// TIA Portal V20 export
TYPE "typeFDoorSignal"
// Safety status of door
// stored: Access Published, IsFailsafeCompliant true, Namespace Safety
   STRUCT
      reqDoorUnlock1 : Bool;   // Cmd Maint Door1 Open Request
      reqDoorUnlock2 : Bool;   // Cmd Maint Door2 Open Request
      reqDoorUnlock3 : Bool;   // Cmd Maint Door3 Open Request
      reqDoorUnlock4 : Bool;   // Cmd Maint Door4 Open Request
      reqDoorUnlock5 : Bool;   // Cmd Maint Door5 Open Request
      reqDoorUnlock6 : Bool;   // Cmd Maint Door6 Open Request
      reqDoorUnlock7 : Bool;   // Cmd Maint Door7 Open Request
      reqDoorUnlock8 : Bool;   // Cmd Maint Door8 Open Request
      reqDoorUnlock9 : Bool;   // Cmd Maint Door9 Open Request
      reqDoorUnlock10 : Bool;   // Cmd Maint Door10 Open Request
   END_STRUCT;
END_TYPE
